TYPE ST_INPUTS_PumpDOL:
STRUCT
	
	Mode:     		E_DeviceMode;
	Command:     E_DeviceState;

END_STRUCT
END_TYPE

(* stored: Version 1.1.0.1, ProductVersion 3.1.4024.12
   DUT ST_INPUTS_PumpDOL: Id {d2230e1b-2d75-410c-92e4-2d5d1dea7555} *)
